# EPICS substitutions: ek9000App/Db/EL3314.substitutions
file EL3314.template
{       pattern
        {
                TERMINAL,

        }
        {
        }
}
